FUNCTION_BLOCK FB_GCLiftPinAxisMoveVelCWServices EXTENDS FB_PackMLModeSet
VAR_INPUT
	Param : ST_GCLiftPinAxisMoveVelParam;
	Ctrl : REFERENCE TO ST_ServiceCtrl;
	Axis_BaseUnit : I_Axis_BaseUnit;

	// The Module assigns a unique ID to this Service instance.
	ResourceOwnerId : T_ResourceOwnerId;
END_VAR

VAR_OUTPUT
	Status : ST_ServiceStatus;
END_VAR

VAR
	_CmdRequestOneShot : R_TRIG;
	_CommandedVelocity : LREAL;
	_VelocityRetriggerPending : BOOL;
END_VAR

PackMLIn := Ctrl.PackMLIn;
SUPER^();

_CmdRequestOneShot(CLK:= PackMLIn.bCommandChangeRequest, Q=> );

// Updata status
Status.PackMLOut := PackMLOut;
IF _CmdRequestOneShot.Q THEN // Acknowledge to upper controller that command received
	Status.ResponseId := Ctrl.RequestId;
END_IF

METHOD PROTECTED H_OnAborted
VAR_INPUT
	bFirstScan	: BOOL;
END_VAR
// Release defensively in case an unexpected transition skipped cleanup.
Axis_BaseUnit.M_ReleaseResource(OwnerId := ResourceOwnerId);

_CommandedVelocity := 0;
_VelocityRetriggerPending := FALSE;
END_METHOD

METHOD PROTECTED H_OnAborting : E_PackMLHookResult
VAR_INPUT
	bFirstScan	: BOOL;
END_VAR

VAR
	bDone : BOOL;
	bError : BOOL;
END_VAR
H_OnAborting := E_PackMLHookResult.Busy;

// A Service that never acquired the Resource must not reset its Owner's Axis.
IF NOT Axis_BaseUnit.M_IsResourceOwner(OwnerId := ResourceOwnerId) THEN
	H_OnAborting := E_PackMLHookResult.Done;
	RETURN;
END_IF

// Withdraw MoveVelocity before resetting the Axis.
Axis_BaseUnit.M_MoveVel(
	OwnerId := ResourceOwnerId,
	Execute := FALSE,
	Direction := MC_Direction.MC_Positive_Direction,
	Velocity := Param.Velocity,
	Acceleration := Param.Acceleration,
	Deceleration := Param.Deceleration);

Axis_BaseUnit.M_Reset(
	OwnerId := ResourceOwnerId,
	Execute := TRUE,
	Done=> bDone, Error=> bError);

IF bDone THEN
	Axis_BaseUnit.M_Reset(
		OwnerId := ResourceOwnerId,
		Execute := FALSE);
	// Keep ownership until the asynchronous Reset has completed.
	Axis_BaseUnit.M_ReleaseResource(OwnerId := ResourceOwnerId);
	H_OnAborting := E_PackMLHookResult.Done;

ELSIF bError THEN
	// A failed Reset is terminal for this Abort sequence; do not remain in Aborting.
	Axis_BaseUnit.M_Reset(
		OwnerId := ResourceOwnerId,
		Execute := FALSE);
	Status.ServiceErrorId := E_GCServiceErrorCode.Error_While_Reset_Axis;
	Axis_BaseUnit.M_ReleaseResource(OwnerId := ResourceOwnerId);
	H_OnAborting := E_PackMLHookResult.Done;
END_IF
END_METHOD

METHOD PROTECTED H_OnClearing : E_PackMLHookResult
VAR_INPUT
	bFirstScan	: BOOL;
END_VAR

VAR
	bServoOn : BOOL;
	bError : BOOL;
	nErrorId : UDINT;
END_VAR
H_OnClearing := E_PackMLHookResult.Done;
END_METHOD

METHOD PROTECTED H_OnComplete
VAR_INPUT
	bFirstScan	: BOOL;
END_VAR
// Completing normally releases first; this is an idempotent safety net.
Axis_BaseUnit.M_ReleaseResource(OwnerId := ResourceOwnerId);
END_METHOD

METHOD PROTECTED H_OnCompleting : E_PackMLHookResult
VAR_INPUT
	bFirstScan	: BOOL;
END_VAR
Axis_BaseUnit.M_MoveVel(
	OwnerId := ResourceOwnerId,
	Execute := FALSE,
	Direction := MC_Direction.MC_Positive_Direction,
	Velocity := Param.Velocity,
	Acceleration := Param.Acceleration,
	Deceleration := Param.Deceleration);

// Release only after the active MoveVelocity request has been withdrawn.
Axis_BaseUnit.M_ReleaseResource(OwnerId := ResourceOwnerId);
H_OnCompleting := E_PackMLHookResult.Done;
END_METHOD

METHOD PROTECTED H_OnExecute : E_PackMLHookResult
VAR_INPUT
	bFirstScan	: BOOL;
END_VAR

VAR
	bError : BOOL;
END_VAR
H_OnExecute := E_PackMLHookResult.Busy;

// Parameters can change while Execute is active, so validate them every scan.
IF (Param.Velocity <= 0) OR (Param.Acceleration < 0) OR (Param.Deceleration < 0) THEN
	Status.ServiceErrorId := E_GCServiceErrorCode.Invalid_Param;
	RequestCommand(E_PackMLCommand.Stop);
	RETURN;
END_IF

// Tc2_MC2 applies new motion parameters on a rising edge of Execute. Keep the
// axis moving while pulsing Execute low for one scan, then retrigger with the
// latest valid velocity and the current acceleration/deceleration values.
IF _VelocityRetriggerPending THEN
	Axis_BaseUnit.M_MoveVel(
		OwnerId := ResourceOwnerId,
		Execute := TRUE,
		Direction := MC_Direction.MC_Positive_Direction,
		Velocity := Param.Velocity,
		Acceleration := Param.Acceleration,
		Deceleration := Param.Deceleration,
		Error=> bError);

	_CommandedVelocity := Param.Velocity;
	_VelocityRetriggerPending := FALSE;

ELSIF Param.Velocity <> _CommandedVelocity THEN
	Axis_BaseUnit.M_MoveVel(
		OwnerId := ResourceOwnerId,
		Execute := FALSE,
		Direction := MC_Direction.MC_Positive_Direction,
		Velocity := Param.Velocity,
		Acceleration := Param.Acceleration,
		Deceleration := Param.Deceleration,
		Error=> bError);

	_VelocityRetriggerPending := TRUE;

ELSE
	Axis_BaseUnit.M_MoveVel(
		OwnerId := ResourceOwnerId,
		Execute := TRUE,
		Direction := MC_Direction.MC_Positive_Direction,
		Velocity := Param.Velocity,
		Acceleration := Param.Acceleration,
		Deceleration := Param.Deceleration,
		Error=> bError);
END_IF

IF bError THEN
	Status.ServiceErrorId := E_GCServiceErrorCode.Axis_Command_Error_During_Execute;
	RequestCommand(E_PackMLCommand.Stop);
END_IF
END_METHOD

METHOD PROTECTED H_OnHeld
VAR_INPUT
	bFirstScan	: BOOL;
END_VAR
// Default action hook intentionally empty. Override in derived FBs when needed.
END_METHOD

METHOD PROTECTED H_OnHolding : E_PackMLHookResult
VAR_INPUT
	bFirstScan	: BOOL;
END_VAR
// Default transient hooks complete immediately; override when work is required.
H_OnHolding := E_PackMLHookResult.Done;
END_METHOD

METHOD PROTECTED H_OnIdle
VAR_INPUT
	bFirstScan	: BOOL;
END_VAR
// Idle Services must not retain a Resource from an earlier operation.
Axis_BaseUnit.M_ReleaseResource(OwnerId := ResourceOwnerId);

_CommandedVelocity := 0;
_VelocityRetriggerPending := FALSE;
END_METHOD

METHOD PROTECTED H_OnResetting : E_PackMLHookResult
VAR_INPUT
	bFirstScan	: BOOL;
END_VAR
Status.ServiceErrorId := E_GCServiceErrorCode.None;

H_OnResetting := E_PackMLHookResult.Done;
END_METHOD

METHOD PROTECTED H_OnStarting : E_PackMLHookResult
VAR_INPUT
	bFirstScan	: BOOL;
END_VAR
H_OnStarting := E_PackMLHookResult.Busy;

// Validate Service-owned data before reserving the shared BaseUnit.
IF Param.Velocity <= 0 THEN
	Status.ServiceErrorId:= E_GCServiceErrorCode.Invalid_Param;
	RequestCommand(E_PackMLCommand.Stop);
	RETURN;
END_IF

IF Param.Acceleration < 0 THEN
	Status.ServiceErrorId:= E_GCServiceErrorCode.Invalid_Param;
	RequestCommand(E_PackMLCommand.Stop);
	RETURN;
END_IF

IF Param.Deceleration < 0 THEN
	Status.ServiceErrorId:= E_GCServiceErrorCode.Invalid_Param;
	RequestCommand(E_PackMLCommand.Stop);
	RETURN;
END_IF

// Resource contention is a failed Start, not a wait condition.
IF NOT Axis_BaseUnit.M_AcquireResource(OwnerId := ResourceOwnerId) THEN
	Status.ServiceErrorId := E_GCServiceErrorCode.Resource_Acquire_Failed_During_Starting;
	RequestCommand(E_PackMLCommand.Stop);
	RETURN;
END_IF

// Physical checks occur only after this Service owns the BaseUnit.
IF Axis_BaseUnit.AxisIsDisabled THEN
	Status.ServiceErrorId:= E_GCServiceErrorCode.Axis_Not_Servo_On_During_Starting;
	RequestCommand(E_PackMLCommand.Abort);
	RETURN;
END_IF

IF Axis_BaseUnit.AxisHasJob THEN
	Status.ServiceErrorId:= E_GCServiceErrorCode.Axis_Is_Busy_During_Starting;
	RequestCommand(E_PackMLCommand.Stop);
	RETURN;
END_IF

_CommandedVelocity := Param.Velocity;
_VelocityRetriggerPending := FALSE;

H_OnStarting := E_PackMLHookResult.Done;
END_METHOD

METHOD PROTECTED H_OnStopped
VAR_INPUT
	bFirstScan	: BOOL;
END_VAR
// Release defensively after every Stop path.
Axis_BaseUnit.M_ReleaseResource(OwnerId := ResourceOwnerId);

_CommandedVelocity := 0;
_VelocityRetriggerPending := FALSE;
END_METHOD

METHOD PROTECTED H_OnStopping : E_PackMLHookResult
VAR_INPUT
	bFirstScan	: BOOL;
END_VAR

VAR
	bDone : BOOL;
	bError : BOOL;
END_VAR
H_OnStopping := E_PackMLHookResult.Busy;

// Resource acquisition failures enter Stopping without owning the Axis.
IF NOT Axis_BaseUnit.M_IsResourceOwner(OwnerId := ResourceOwnerId) THEN
	H_OnStopping := E_PackMLHookResult.Done;
	RETURN;
END_IF

// Withdraw MoveVelocity before issuing the physical Stop.
Axis_BaseUnit.M_MoveVel(
	OwnerId := ResourceOwnerId,
	Execute := FALSE,
	Direction := MC_Direction.MC_Positive_Direction,
	Velocity := Param.Velocity,
	Acceleration := Param.Acceleration,
	Deceleration := Param.Deceleration);

Axis_BaseUnit.M_Stop(
	OwnerId := ResourceOwnerId,
	Execute := TRUE,
	Deceleration:= Param.Deceleration,
	Done=> bDone, Error=> bError);

IF bDone THEN
	Axis_BaseUnit.M_Stop(
		OwnerId := ResourceOwnerId,
		Execute := FALSE,
		Deceleration:= Param.Deceleration);
	// Ownership is released only after the asynchronous Stop has completed.
	Axis_BaseUnit.M_ReleaseResource(OwnerId := ResourceOwnerId);
	H_OnStopping := E_PackMLHookResult.Done;

ELSIF bError THEN
	// Throw up error
	Status.ServiceErrorId := E_GCServiceErrorCode.Error_While_Stop_Axis;

	Axis_BaseUnit.M_Stop(
		OwnerId := ResourceOwnerId,
		Execute := FALSE,
		Deceleration:= Param.Deceleration);

	RequestCommand(E_PackMLCommand.Abort);
END_IF
END_METHOD

METHOD PROTECTED H_OnSuspended
VAR_INPUT
	bFirstScan	: BOOL;
END_VAR
// Default action hook intentionally empty. Override in derived FBs when needed.
END_METHOD

METHOD PROTECTED H_OnSuspending : E_PackMLHookResult
VAR_INPUT
	bFirstScan	: BOOL;
END_VAR
// Default transient hooks complete immediately; override when work is required.
H_OnSuspending := E_PackMLHookResult.Done;
END_METHOD

METHOD PROTECTED H_OnUndefined : E_PackMLHookResult
VAR_INPUT
	bFirstScan	: BOOL;
END_VAR
// The base FB leaves Undefined immediately unless a derived FB delays startup.
H_OnUndefined := E_PackMLHookResult.Done;
END_METHOD

METHOD PROTECTED H_OnUnholding : E_PackMLHookResult
VAR_INPUT
	bFirstScan	: BOOL;
END_VAR
// Default transient hooks complete immediately; override when work is required.
H_OnUnholding := E_PackMLHookResult.Done;
END_METHOD

METHOD PROTECTED H_OnUnsuspending : E_PackMLHookResult
VAR_INPUT
	bFirstScan	: BOOL;
END_VAR
// Default transient hooks complete immediately; override when work is required.
H_OnUnsuspending := E_PackMLHookResult.Done;
END_METHOD

END_FUNCTION_BLOCK

(* stored: Version 1.1.0.1, ProductVersion 3.1.4026.18
   POU FB_GCLiftPinAxisMoveVelCWServices: Id {a1c00001-6b2c-4d3e-8f90-a1c000000001}, SpecialFunc None
   Folder StateAction: Id {a1c00002-6b2c-4d3e-8f90-a1c000000002}
   Method H_OnAborted: Id {a1c00003-6b2c-4d3e-8f90-a1c000000003}
   Method H_OnAborting: Id {a1c00004-6b2c-4d3e-8f90-a1c000000004}
   Method H_OnClearing: Id {a1c00005-6b2c-4d3e-8f90-a1c000000005}
   Method H_OnComplete: Id {a1c00006-6b2c-4d3e-8f90-a1c000000006}
   Method H_OnCompleting: Id {a1c00007-6b2c-4d3e-8f90-a1c000000007}
   Method H_OnExecute: Id {a1c00008-6b2c-4d3e-8f90-a1c000000008}
   Method H_OnHeld: Id {a1c00009-6b2c-4d3e-8f90-a1c000000009}
   Method H_OnHolding: Id {a1c0000a-6b2c-4d3e-8f90-a1c00000000a}
   Method H_OnIdle: Id {a1c0000b-6b2c-4d3e-8f90-a1c00000000b}
   Method H_OnResetting: Id {a1c0000c-6b2c-4d3e-8f90-a1c00000000c}
   Method H_OnStarting: Id {a1c0000d-6b2c-4d3e-8f90-a1c00000000d}
   Method H_OnStopped: Id {a1c0000e-6b2c-4d3e-8f90-a1c00000000e}
   Method H_OnStopping: Id {a1c0000f-6b2c-4d3e-8f90-a1c00000000f}
   Method H_OnSuspended: Id {a1c00010-6b2c-4d3e-8f90-a1c000000010}
   Method H_OnSuspending: Id {a1c00011-6b2c-4d3e-8f90-a1c000000011}
   Method H_OnUndefined: Id {a1c00012-6b2c-4d3e-8f90-a1c000000012}
   Method H_OnUnholding: Id {a1c00013-6b2c-4d3e-8f90-a1c000000013}
   Method H_OnUnsuspending: Id {a1c00014-6b2c-4d3e-8f90-a1c000000014} *)
